TYPE "Type_Output"
VERSION : 0.1
   STRUCT
      val_in : Real;
      val_norm : Real;
      val_scaled : Real;
      out_dig1 : Bool;
      out_dig2 : Bool;
      out_analog1 : DInt;
      out_analog2 : DInt;
      flagao : Bool;
      indasse : Int := -1;
      enab : Bool;
      preset : Bool;
      preval : Real;
      preind2 : Int;
   END_STRUCT;

END_TYPE

